TYPE IO_Typ :
STRUCT
	In:IO_In_Typ;
	Out:IO_Out_Typ;
	EncoderRW:Encoder_Typ;
	//RwInverter:ST_BasicInverter;
END_STRUCT
END_TYPE

(* stored: Version 1.1.0.1, ProductVersion 3.1.4024.3
   DUT IO_Typ: Id {50458ce5-806d-458e-ac25-a91f59162c16} *)
